% RSLogix 500 project CCHOUTSIDE BS_BAK004.RSS, saved by version 11.00.00.00 %
PROJECT "FMCBIN"    % processor: MicroLogix 1200 %

PROGRAM FILES
  LAD 2   45 rungs
  LAD 3   24 rungs
  LAD 4   21 rungs

DATA FILES
  O0 OUTPUT  5 elements
  I1 INPUT  6 elements
  S2 STATUS  66 elements
  B3 BINARY  5 elements
  T4 TIMER  28 elements
  C5 COUNTER  10 elements
  R6 CONTROL  1 elements
  N7 INTEGER  6 elements
  F8 FLOAT  1 elements

LADDER 2
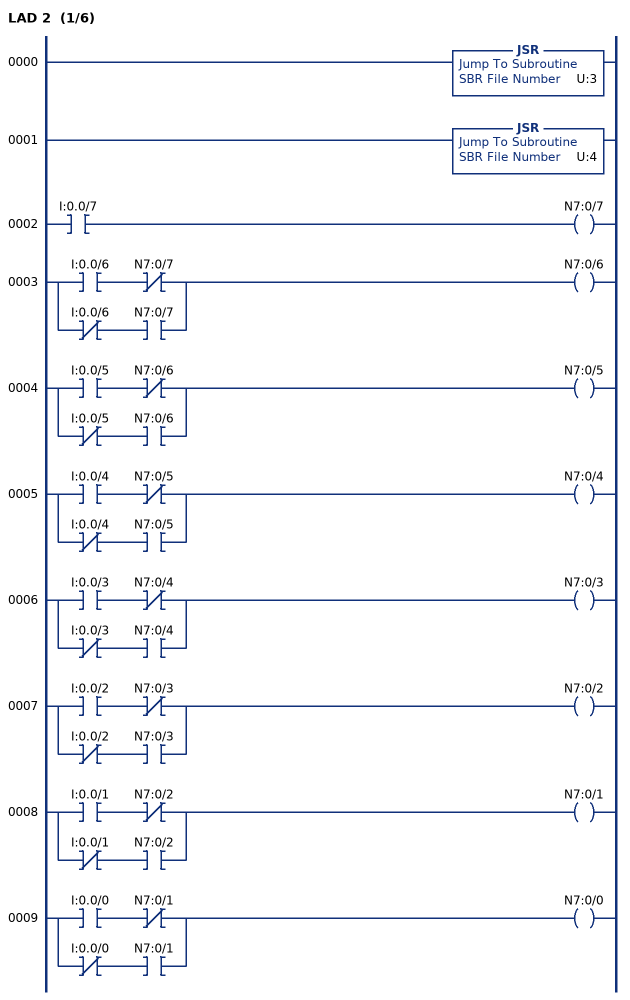
% Rung: 0 %
SOR JSR U:3 EOR
% Rung: 1 %
SOR JSR U:4 EOR
% Rung: 2 %
SOR XIC I:0.0/7 OTE N7:0/7 EOR
% Rung: 3 %
SOR BST XIC I:0.0/6 XIO N7:0/7 NXB XIO I:0.0/6 XIC N7:0/7 BND OTE N7:0/6 EOR
% Rung: 4 %
SOR BST XIC I:0.0/5 XIO N7:0/6 NXB XIO I:0.0/5 XIC N7:0/6 BND OTE N7:0/5 EOR
% Rung: 5 %
SOR BST XIC I:0.0/4 XIO N7:0/5 NXB XIO I:0.0/4 XIC N7:0/5 BND OTE N7:0/4 EOR
% Rung: 6 %
SOR BST XIC I:0.0/3 XIO N7:0/4 NXB XIO I:0.0/3 XIC N7:0/4 BND OTE N7:0/3 EOR
% Rung: 7 %
SOR BST XIC I:0.0/2 XIO N7:0/3 NXB XIO I:0.0/2 XIC N7:0/3 BND OTE N7:0/2 EOR
% Rung: 8 %
SOR BST XIC I:0.0/1 XIO N7:0/2 NXB XIO I:0.0/1 XIC N7:0/2 BND OTE N7:0/1 EOR
% Rung: 9 %
SOR BST XIC I:0.0/0 XIO N7:0/1 NXB XIO I:0.0/0 XIC N7:0/1 BND OTE N7:0/0 EOR

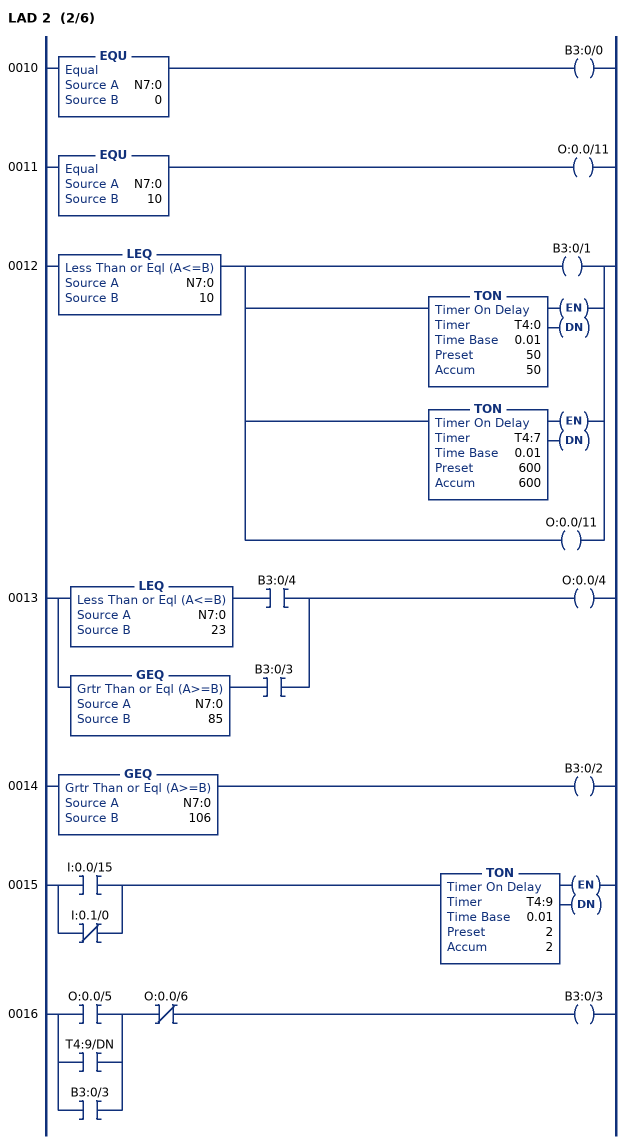
% Rung: 10 %
SOR EQU N7:0 0 OTE B3:0/0 EOR
% Rung: 11 %
SOR EQU N7:0 10 OTE O:0.0/11 EOR
% Rung: 12 %
SOR LEQ N7:0 10 BST OTE B3:0/1 NXB TON T4:0 0.01 50 50 NXB BST TON T4:7 0.01 600 600 NXB OTE O:0.0/11 BND BND EOR
% Rung: 13 %
SOR BST LEQ N7:0 23 XIC B3:0/4 NXB GEQ N7:0 85 XIC B3:0/3 BND OTE O:0.0/4 EOR
% Rung: 14 %
SOR GEQ N7:0 106 OTE B3:0/2 EOR
% Rung: 15 %
SOR BST XIC I:0.0/15 NXB XIO I:0.1/0 BND TON T4:9 0.01 2 2 EOR
% Rung: 16 %
SOR BST XIC O:0.0/5 NXB XIC T4:9/DN NXB XIC B3:0/3 BND XIO O:0.0/6 OTE B3:0/3 EOR

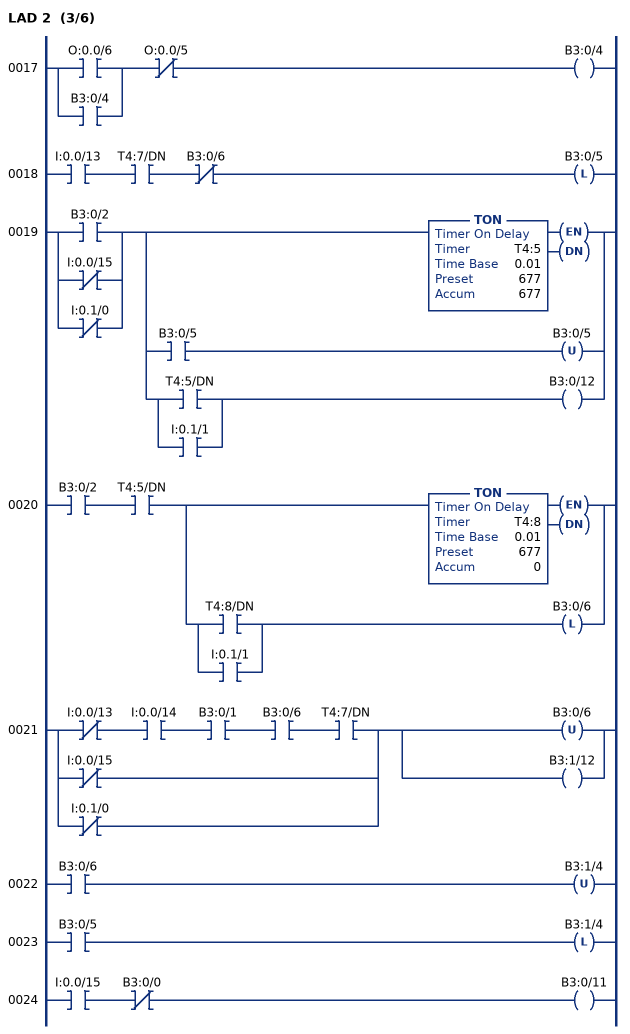
% Rung: 17 %
SOR BST XIC O:0.0/6 NXB XIC B3:0/4 BND XIO O:0.0/5 OTE B3:0/4 EOR
% Rung: 18 %
SOR XIC I:0.0/13 XIC T4:7/DN XIO B3:0/6 OTL B3:0/5 EOR
% Rung: 19 %
SOR BST XIC B3:0/2 NXB XIO I:0.0/15 NXB XIO I:0.1/0 BND BST TON T4:5 0.01 677 677 NXB XIC B3:0/5 OTU B3:0/5 NXB BST XIC T4:5/DN NXB XIC I:0.1/1 BND OTE B3:0/12 BND EOR
% Rung: 20 %
SOR XIC B3:0/2 XIC T4:5/DN BST TON T4:8 0.01 677 0 NXB BST XIC T4:8/DN NXB XIC I:0.1/1 BND OTL B3:0/6 BND EOR
% Rung: 21 %
SOR BST XIO I:0.0/13 XIC I:0.0/14 XIC B3:0/1 XIC B3:0/6 XIC T4:7/DN NXB BST XIO I:0.0/15 NXB XIO I:0.1/0 BND BND BST OTU B3:0/6 NXB OTE B3:1/12 BND EOR
% Rung: 22 %
SOR XIC B3:0/6 OTU B3:1/4 EOR
% Rung: 23 %
SOR XIC B3:0/5 OTL B3:1/4 EOR
% Rung: 24 %
SOR XIC I:0.0/15 XIO B3:0/0 OTE B3:0/11 EOR

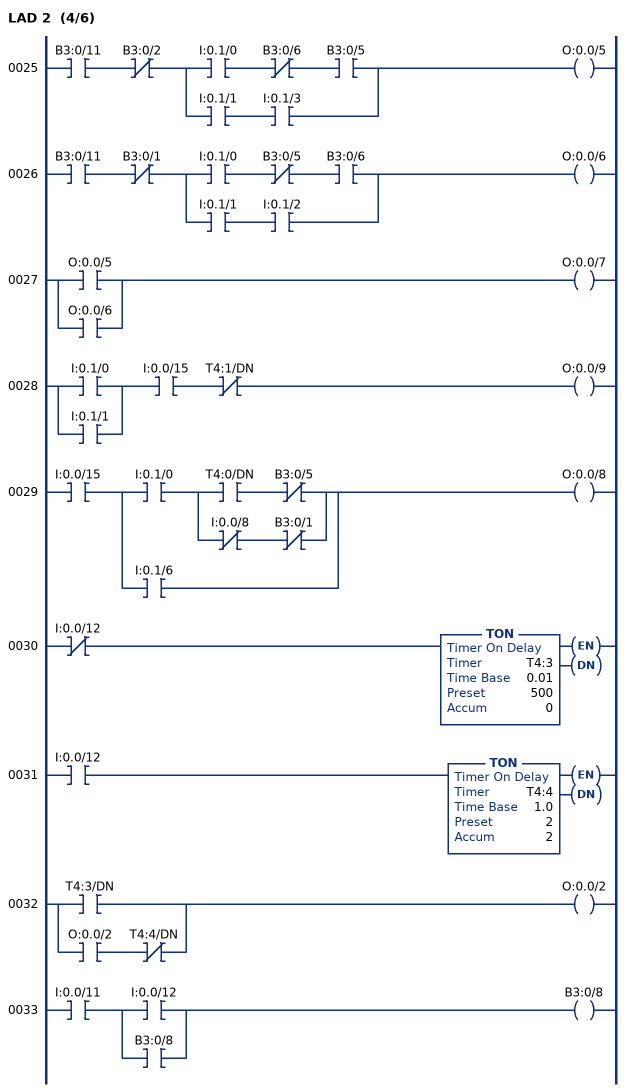
% Rung: 25 %
SOR XIC B3:0/11 XIO B3:0/2 BST XIC I:0.1/0 XIO B3:0/6 XIC B3:0/5 NXB XIC I:0.1/1 XIC I:0.1/3 BND OTE O:0.0/5 EOR
% Rung: 26 %
SOR XIC B3:0/11 XIO B3:0/1 BST XIC I:0.1/0 XIO B3:0/5 XIC B3:0/6 NXB XIC I:0.1/1 XIC I:0.1/2 BND OTE O:0.0/6 EOR
% Rung: 27 %
SOR BST XIC O:0.0/5 NXB XIC O:0.0/6 BND OTE O:0.0/7 EOR
% Rung: 28 %
SOR BST XIC I:0.1/0 NXB XIC I:0.1/1 BND XIC I:0.0/15 XIO T4:1/DN OTE O:0.0/9 EOR
% Rung: 29 %
SOR XIC I:0.0/15 BST XIC I:0.1/0 BST XIC T4:0/DN XIO B3:0/5 NXB XIO I:0.0/8 XIO B3:0/1 BND NXB XIC I:0.1/6 BND OTE O:0.0/8 EOR
% Rung: 30 %
SOR XIO I:0.0/12 TON T4:3 0.01 500 0 EOR
% Rung: 31 %
SOR XIC I:0.0/12 TON T4:4 1.0 2 2 EOR
% Rung: 32 %
SOR BST XIC T4:3/DN NXB XIC O:0.0/2 XIO T4:4/DN BND OTE O:0.0/2 EOR
% Rung: 33 %
SOR XIC I:0.0/11 BST XIC I:0.0/12 NXB XIC B3:0/8 BND OTE B3:0/8 EOR

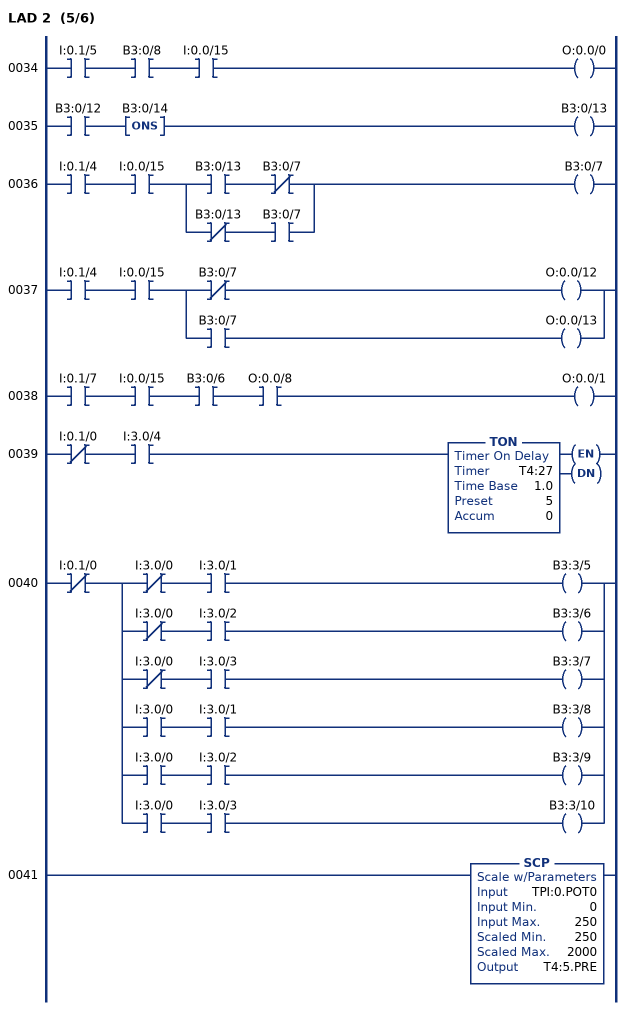
% Rung: 34 %
SOR XIC I:0.1/5 XIC B3:0/8 XIC I:0.0/15 OTE O:0.0/0 EOR
% Rung: 35 %
SOR XIC B3:0/12 ONS B3:0/14 OTE B3:0/13 EOR
% Rung: 36 %
SOR XIC I:0.1/4 XIC I:0.0/15 BST XIC B3:0/13 XIO B3:0/7 NXB XIO B3:0/13 XIC B3:0/7 BND OTE B3:0/7 EOR
% Rung: 37 %
SOR XIC I:0.1/4 XIC I:0.0/15 BST XIO B3:0/7 OTE O:0.0/12 NXB XIC B3:0/7 OTE O:0.0/13 BND EOR
% Rung: 38 %
SOR XIC I:0.1/7 XIC I:0.0/15 XIC B3:0/6 XIC O:0.0/8 OTE O:0.0/1 EOR
% Rung: 39 %
SOR XIO I:0.1/0 XIC I:3.0/4 TON T4:27 1.0 5 0 EOR
% Rung: 40 %
SOR XIO I:0.1/0 BST XIO I:3.0/0 XIC I:3.0/1 OTE B3:3/5 NXB XIO I:3.0/0 XIC I:3.0/2 OTE B3:3/6 NXB XIO I:3.0/0 XIC I:3.0/3 OTE B3:3/7 NXB XIC I:3.0/0 XIC I:3.0/1 OTE B3:3/8 NXB XIC I:3.0/0 XIC I:3.0/2 OTE B3:3/9 NXB XIC I:3.0/0 XIC I:3.0/3 OTE B3:3/10 BND EOR
% Rung: 41 %
SOR SCP TPI:0.POT0 0 250 250 2000 T4:5.PRE EOR

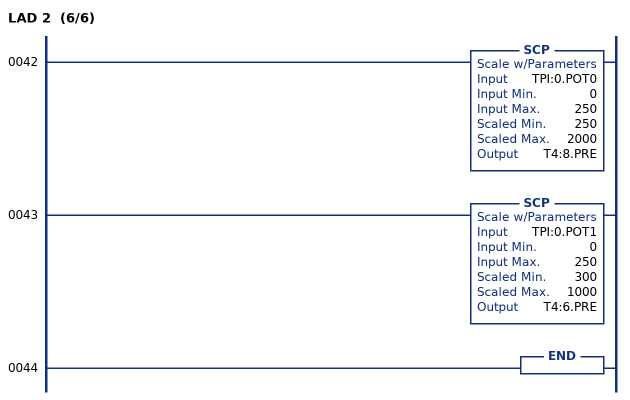
% Rung: 42 %
SOR SCP TPI:0.POT0 0 250 250 2000 T4:8.PRE EOR
% Rung: 43 %
SOR SCP TPI:0.POT1 0 250 300 1000 T4:6.PRE EOR
% Rung: 44 %
SOR END EOR

LADDER 3
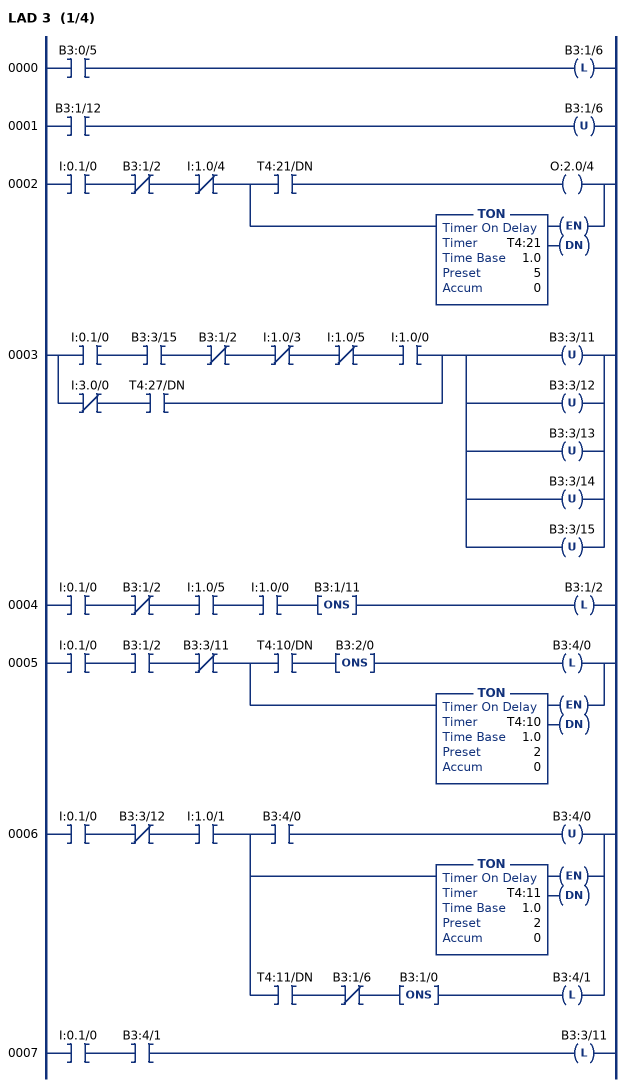
% Rung: 0 %
SOR XIC B3:0/5 OTL B3:1/6 EOR
% Rung: 1 %
SOR XIC B3:1/12 OTU B3:1/6 EOR
% Rung: 2 %
SOR XIC I:0.1/0 XIO B3:1/2 XIO I:1.0/4 BST XIC T4:21/DN OTE O:2.0/4 NXB TON T4:21 1.0 5 0 BND EOR
% Rung: 3 %
SOR BST XIC I:0.1/0 XIC B3:3/15 XIO B3:1/2 XIO I:1.0/3 XIO I:1.0/5 XIC I:1.0/0 NXB XIO I:3.0/0 XIC T4:27/DN BND BST OTU B3:3/11 NXB OTU B3:3/12 NXB OTU B3:3/13 NXB OTU B3:3/14 NXB OTU B3:3/15 BND EOR
% Rung: 4 %
SOR XIC I:0.1/0 XIO B3:1/2 XIC I:1.0/5 XIC I:1.0/0 ONS B3:1/11 OTL B3:1/2 EOR
% Rung: 5 %
SOR XIC I:0.1/0 XIC B3:1/2 XIO B3:3/11 BST XIC T4:10/DN ONS B3:2/0 OTL B3:4/0 NXB TON T4:10 1.0 2 0 BND EOR
% Rung: 6 %
SOR XIC I:0.1/0 XIO B3:3/12 XIC I:1.0/1 BST XIC B3:4/0 OTU B3:4/0 NXB TON T4:11 1.0 2 0 NXB XIC T4:11/DN XIO B3:1/6 ONS B3:1/0 OTL B3:4/1 BND EOR
% Rung: 7 %
SOR XIC I:0.1/0 XIC B3:4/1 OTL B3:3/11 EOR

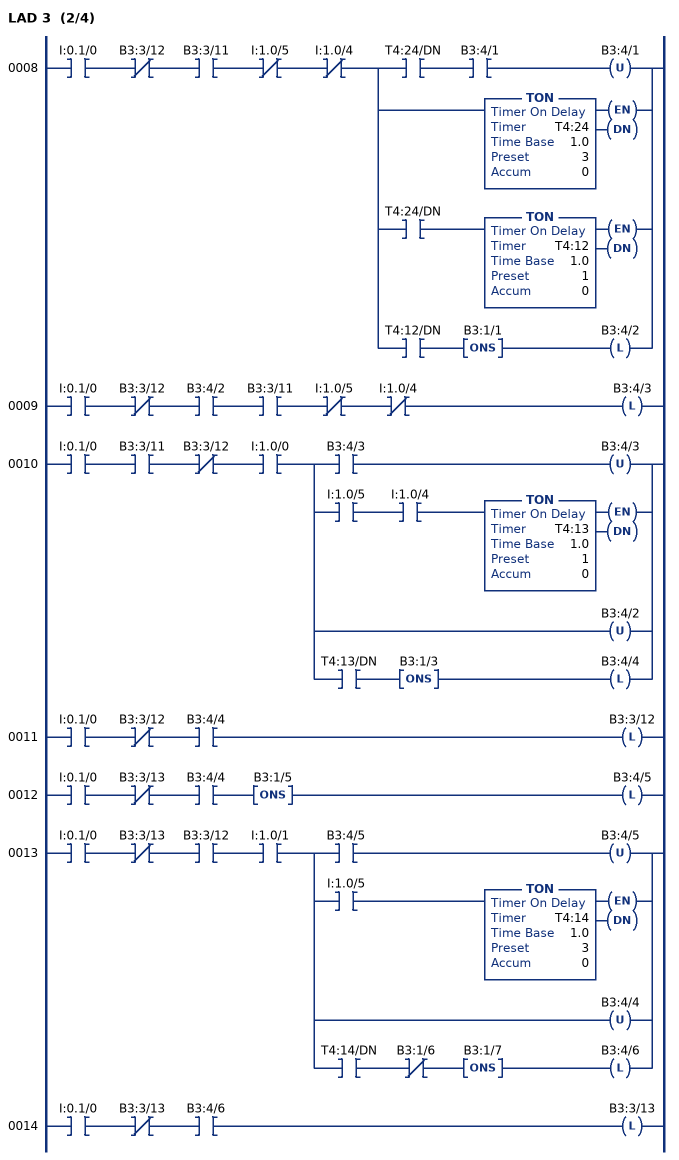
% Rung: 8 %
SOR XIC I:0.1/0 XIO B3:3/12 XIC B3:3/11 XIO I:1.0/5 XIO I:1.0/4 BST XIC T4:24/DN XIC B3:4/1 OTU B3:4/1 NXB TON T4:24 1.0 3 0 NXB XIC T4:24/DN TON T4:12 1.0 1 0 NXB XIC T4:12/DN ONS B3:1/1 OTL B3:4/2 BND EOR
% Rung: 9 %
SOR XIC I:0.1/0 XIO B3:3/12 XIC B3:4/2 XIC B3:3/11 XIO I:1.0/5 XIO I:1.0/4 OTL B3:4/3 EOR
% Rung: 10 %
SOR XIC I:0.1/0 XIC B3:3/11 XIO B3:3/12 XIC I:1.0/0 BST XIC B3:4/3 OTU B3:4/3 NXB XIC I:1.0/5 XIC I:1.0/4 TON T4:13 1.0 1 0 NXB OTU B3:4/2 NXB XIC T4:13/DN ONS B3:1/3 OTL B3:4/4 BND EOR
% Rung: 11 %
SOR XIC I:0.1/0 XIO B3:3/12 XIC B3:4/4 OTL B3:3/12 EOR
% Rung: 12 %
SOR XIC I:0.1/0 XIO B3:3/13 XIC B3:4/4 ONS B3:1/5 OTL B3:4/5 EOR
% Rung: 13 %
SOR XIC I:0.1/0 XIO B3:3/13 XIC B3:3/12 XIC I:1.0/1 BST XIC B3:4/5 OTU B3:4/5 NXB XIC I:1.0/5 TON T4:14 1.0 3 0 NXB OTU B3:4/4 NXB XIC T4:14/DN XIO B3:1/6 ONS B3:1/7 OTL B3:4/6 BND EOR
% Rung: 14 %
SOR XIC I:0.1/0 XIO B3:3/13 XIC B3:4/6 OTL B3:3/13 EOR

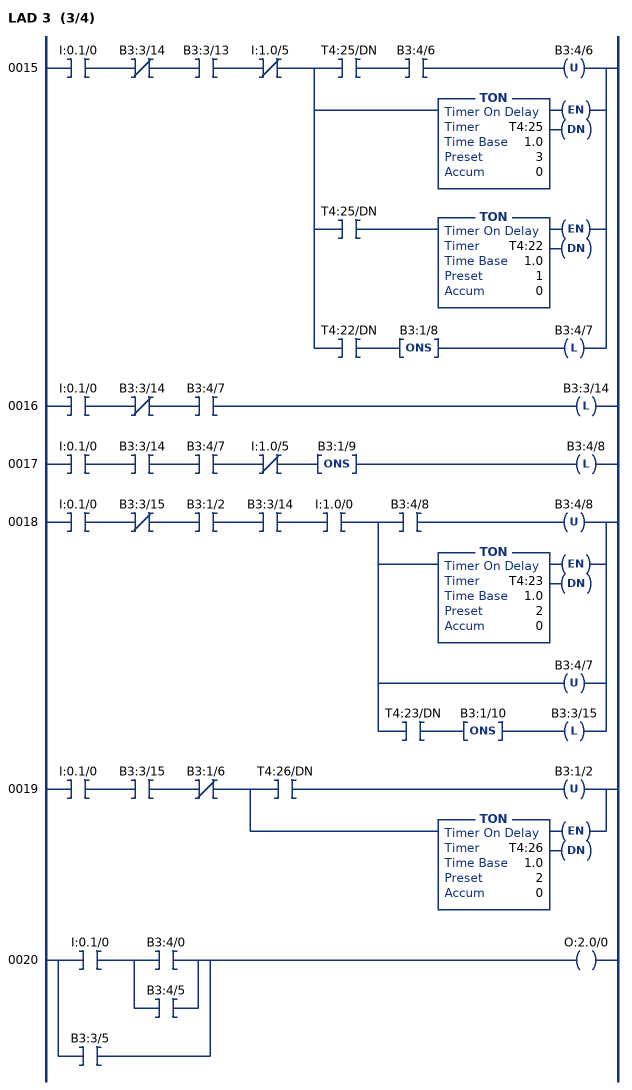
% Rung: 15 %
SOR XIC I:0.1/0 XIO B3:3/14 XIC B3:3/13 XIO I:1.0/5 BST XIC T4:25/DN XIC B3:4/6 OTU B3:4/6 NXB TON T4:25 1.0 3 0 NXB XIC T4:25/DN TON T4:22 1.0 1 0 NXB XIC T4:22/DN ONS B3:1/8 OTL B3:4/7 BND EOR
% Rung: 16 %
SOR XIC I:0.1/0 XIO B3:3/14 XIC B3:4/7 OTL B3:3/14 EOR
% Rung: 17 %
SOR XIC I:0.1/0 XIC B3:3/14 XIC B3:4/7 XIO I:1.0/5 ONS B3:1/9 OTL B3:4/8 EOR
% Rung: 18 %
SOR XIC I:0.1/0 XIO B3:3/15 XIC B3:1/2 XIC B3:3/14 XIC I:1.0/0 BST XIC B3:4/8 OTU B3:4/8 NXB TON T4:23 1.0 2 0 NXB OTU B3:4/7 NXB XIC T4:23/DN ONS B3:1/10 OTL B3:3/15 BND EOR
% Rung: 19 %
SOR XIC I:0.1/0 XIC B3:3/15 XIO B3:1/6 BST XIC T4:26/DN OTU B3:1/2 NXB TON T4:26 1.0 2 0 BND EOR
% Rung: 20 %
SOR BST XIC I:0.1/0 BST XIC B3:4/0 NXB XIC B3:4/5 BND NXB XIC B3:3/5 BND OTE O:2.0/0 EOR

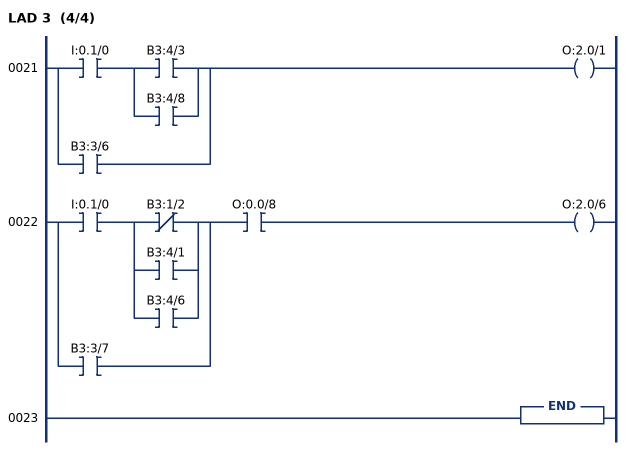
% Rung: 21 %
SOR BST XIC I:0.1/0 BST XIC B3:4/3 NXB XIC B3:4/8 BND NXB XIC B3:3/6 BND OTE O:2.0/1 EOR
% Rung: 22 %
SOR BST XIC I:0.1/0 BST XIO B3:1/2 NXB XIC B3:4/1 NXB XIC B3:4/6 BND NXB XIC B3:3/7 BND XIC O:0.0/8 OTE O:2.0/6 EOR
% Rung: 23 %
SOR END EOR

LADDER 4
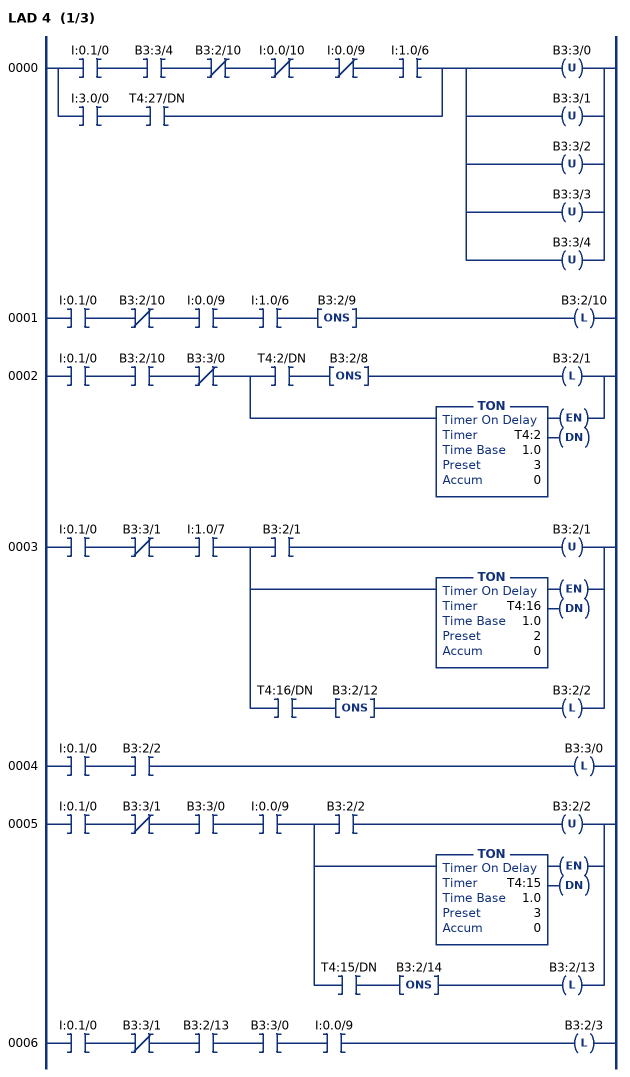
% Rung: 0 %
SOR BST XIC I:0.1/0 XIC B3:3/4 XIO B3:2/10 XIO I:0.0/10 XIO I:0.0/9 XIC I:1.0/6 NXB XIC I:3.0/0 XIC T4:27/DN BND BST OTU B3:3/0 NXB OTU B3:3/1 NXB OTU B3:3/2 NXB OTU B3:3/3 NXB OTU B3:3/4 BND EOR
% Rung: 1 %
SOR XIC I:0.1/0 XIO B3:2/10 XIC I:0.0/9 XIC I:1.0/6 ONS B3:2/9 OTL B3:2/10 EOR
% Rung: 2 %
SOR XIC I:0.1/0 XIC B3:2/10 XIO B3:3/0 BST XIC T4:2/DN ONS B3:2/8 OTL B3:2/1 NXB TON T4:2 1.0 3 0 BND EOR
% Rung: 3 %
SOR XIC I:0.1/0 XIO B3:3/1 XIC I:1.0/7 BST XIC B3:2/1 OTU B3:2/1 NXB TON T4:16 1.0 2 0 NXB XIC T4:16/DN ONS B3:2/12 OTL B3:2/2 BND EOR
% Rung: 4 %
SOR XIC I:0.1/0 XIC B3:2/2 OTL B3:3/0 EOR
% Rung: 5 %
SOR XIC I:0.1/0 XIO B3:3/1 XIC B3:3/0 XIC I:0.0/9 BST XIC B3:2/2 OTU B3:2/2 NXB TON T4:15 1.0 3 0 NXB XIC T4:15/DN ONS B3:2/14 OTL B3:2/13 BND EOR
% Rung: 6 %
SOR XIC I:0.1/0 XIO B3:3/1 XIC B3:2/13 XIC B3:3/0 XIC I:0.0/9 OTL B3:2/3 EOR

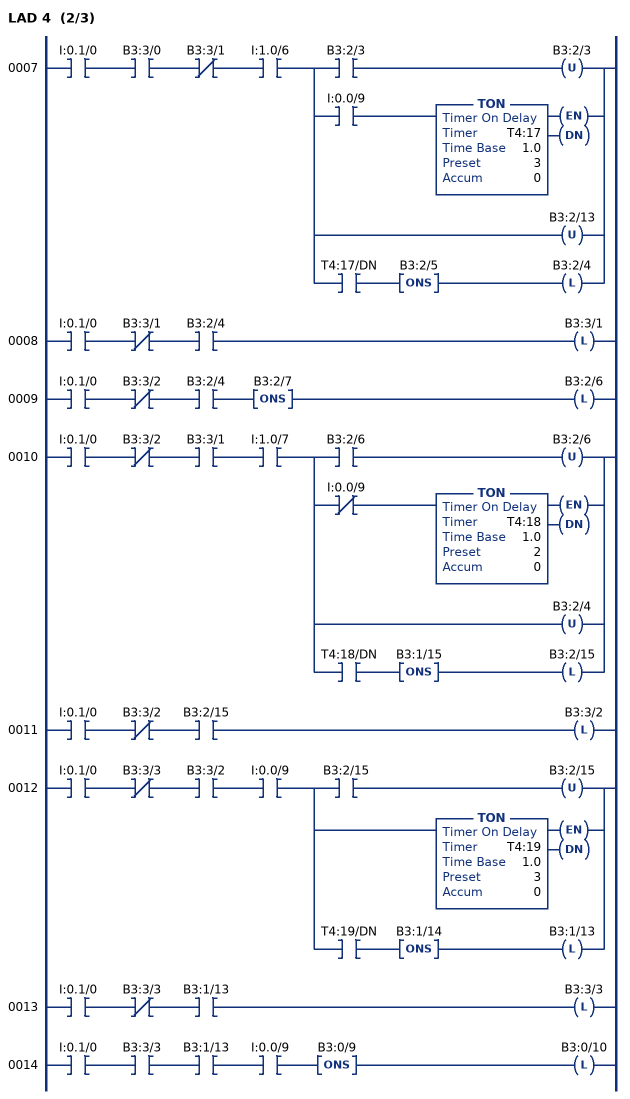
% Rung: 7 %
SOR XIC I:0.1/0 XIC B3:3/0 XIO B3:3/1 XIC I:1.0/6 BST XIC B3:2/3 OTU B3:2/3 NXB XIC I:0.0/9 TON T4:17 1.0 3 0 NXB OTU B3:2/13 NXB XIC T4:17/DN ONS B3:2/5 OTL B3:2/4 BND EOR
% Rung: 8 %
SOR XIC I:0.1/0 XIO B3:3/1 XIC B3:2/4 OTL B3:3/1 EOR
% Rung: 9 %
SOR XIC I:0.1/0 XIO B3:3/2 XIC B3:2/4 ONS B3:2/7 OTL B3:2/6 EOR
% Rung: 10 %
SOR XIC I:0.1/0 XIO B3:3/2 XIC B3:3/1 XIC I:1.0/7 BST XIC B3:2/6 OTU B3:2/6 NXB XIO I:0.0/9 TON T4:18 1.0 2 0 NXB OTU B3:2/4 NXB XIC T4:18/DN ONS B3:1/15 OTL B3:2/15 BND EOR
% Rung: 11 %
SOR XIC I:0.1/0 XIO B3:3/2 XIC B3:2/15 OTL B3:3/2 EOR
% Rung: 12 %
SOR XIC I:0.1/0 XIO B3:3/3 XIC B3:3/2 XIC I:0.0/9 BST XIC B3:2/15 OTU B3:2/15 NXB TON T4:19 1.0 3 0 NXB XIC T4:19/DN ONS B3:1/14 OTL B3:1/13 BND EOR
% Rung: 13 %
SOR XIC I:0.1/0 XIO B3:3/3 XIC B3:1/13 OTL B3:3/3 EOR
% Rung: 14 %
SOR XIC I:0.1/0 XIC B3:3/3 XIC B3:1/13 XIC I:0.0/9 ONS B3:0/9 OTL B3:0/10 EOR

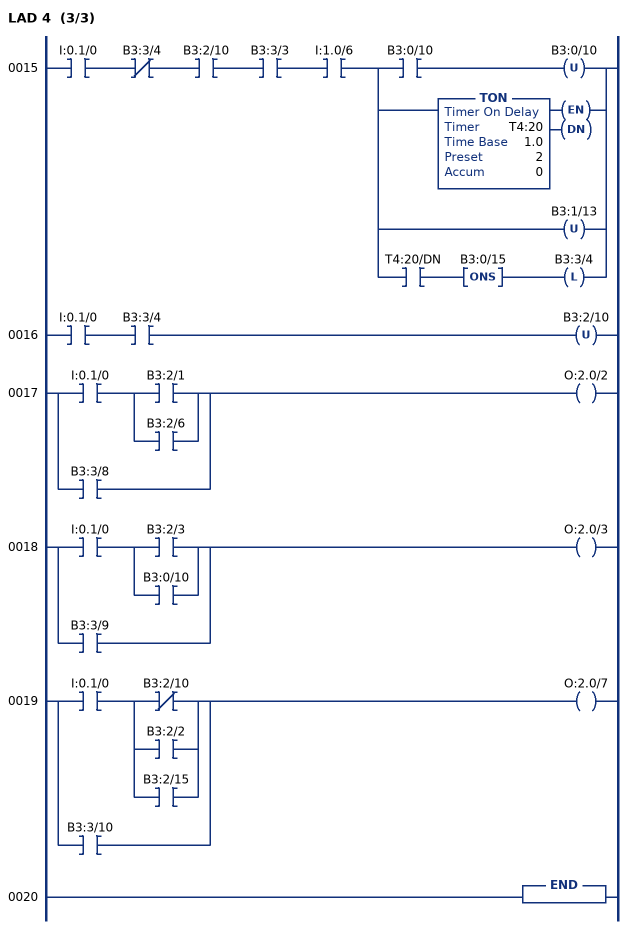
% Rung: 15 %
SOR XIC I:0.1/0 XIO B3:3/4 XIC B3:2/10 XIC B3:3/3 XIC I:1.0/6 BST XIC B3:0/10 OTU B3:0/10 NXB TON T4:20 1.0 2 0 NXB OTU B3:1/13 NXB XIC T4:20/DN ONS B3:0/15 OTL B3:3/4 BND EOR
% Rung: 16 %
SOR XIC I:0.1/0 XIC B3:3/4 OTU B3:2/10 EOR
% Rung: 17 %
SOR BST XIC I:0.1/0 BST XIC B3:2/1 NXB XIC B3:2/6 BND NXB XIC B3:3/8 BND OTE O:2.0/2 EOR
% Rung: 18 %
SOR BST XIC I:0.1/0 BST XIC B3:2/3 NXB XIC B3:0/10 BND NXB XIC B3:3/9 BND OTE O:2.0/3 EOR
% Rung: 19 %
SOR BST XIC I:0.1/0 BST XIO B3:2/10 NXB XIC B3:2/2 NXB XIC B3:2/15 BND NXB XIC B3:3/10 BND OTE O:2.0/7 EOR
% Rung: 20 %
SOR END EOR

DATA TABLE (non-zero values as saved)
DATA B3
% B3:0 % 0X511A 0X1010 0X0800 0X0000 0X0000
DATA T4
% .PRE .ACC %
% T4:0 % 50 50
% T4:1 % 1 0
% T4:2 % 3 0
% T4:3 % 500 0
% T4:4 % 2 2
% T4:5 % 677 677
% T4:6 % 692 0
% T4:7 % 600 600
% T4:8 % 677 0
% T4:9 % 2 2
% T4:10 % 2 0
% T4:11 % 2 0
% T4:12 % 1 0
% T4:13 % 1 0
% T4:14 % 3 0
% T4:15 % 3 0
% T4:16 % 2 0
% T4:17 % 3 0
% T4:18 % 2 0
% T4:19 % 3 0
% T4:20 % 2 0
% T4:21 % 5 0
% T4:22 % 1 0
% T4:23 % 2 0
% T4:24 % 3 0
% T4:25 % 3 0
% T4:26 % 2 0
% T4:27 % 5 0
DATA C5
% .PRE .ACC %
% C5:0 % 2 3
DATA N7
% N7:0 % 10 0 0 0 0 0
